// TIA Portal V20 export
// export: Created 2026-04-11T06:02:29.7304314Z, ExportSetting WithDefaults, DisplayName Totally Integrated Automation Portal, DisplayVersion V20, DisplayName TIA Portal Openness, DisplayVersion V20, DisplayName TIA Portal Version Control Interface, DisplayVersion V20, DisplayName STEP 7 Professional, DisplayVersion V20, DisplayName STEP 7 Safety, DisplayVersion V20, DisplayName WinCC Basic/Comfort/Advanced, DisplayVersion V20, DisplayName WinCC Unified, DisplayVersion V20
TYPE "udtHMI_Valve3WayControl"
// stored: IsFailsafeCompliant false
   STRUCT
      iMode : Int;   // Current mode code
      iErrorCode { ExternalWritable := 'False'} : Int;   // Error code
      iStatus { ExternalWritable := 'False'} : Int;   // HMI status
      bPB_ResetError : Bool;   // Reset error button
      bPB_Home : Bool;   // PB move to Home in manual mode
      bPB_Work : Bool;   // PB move to Work in manual mode
      bPB_Stop : Bool;   // PB stop in the intermediate position
      bPBEN_ResetError { ExternalWritable := 'False'} : Bool;   // Reset button enable
      bPBEN_Home { ExternalWritable := 'False'} : Bool;   // PB Home button enable
      bPBEN_Work { ExternalWritable := 'False'} : Bool;   // PB Work button enable
      bPBEN_Stop { ExternalWritable := 'False'} : Bool;   // PB Stop button enable
      bHomeOn { ExternalWritable := 'False'} : Bool;   // Go to Home
      bWorkOn { ExternalWritable := 'False'} : Bool;   // Go to Work
      bSignalHome { ExternalWritable := 'False'} : Bool;   // Home feedback
      bSignalWork { ExternalWritable := 'False'} : Bool;   // Work feedback
      bInterlock { ExternalWritable := 'False'} : Bool;   // Interlock is on
      bError { ExternalWritable := 'False'} : Bool;   // Error status
   END_STRUCT;
END_TYPE
